// TIA Portal V18 export
TYPE "UDT_OAT"
// stored: IsFailsafeCompliant false
   STRUCT
      rOAT_PLC_IO : Real;
      rOAT_WeatherStation : Real;
      rOAT_Boilers : Real;
      rOAT_Actual : Real;
   END_STRUCT;
END_TYPE
